// TIA Portal V17 export
// export: Created 2025-03-05T08:03:12.1647965Z, ExportSetting WithDefaults, DisplayName Totally Integrated Automation Portal, DisplayVersion V17 Update 8, DisplayName TIA Portal Openness, DisplayVersion V17 Update 8, DisplayName TIA Portal Version Control Interface, DisplayVersion V17, DisplayName SINAMICS Startdrive Advanced, DisplayVersion V17 SP2, DisplayName SINAMICS Startdrive G110M, G120, G120C, G120D, G120P, G115D, DisplayVersion V17 SP2, DisplayName SINAMICS Startdrive G130, G150, S120, S150, SINAMICS MV, S210, DisplayVersion V17 SP2, DisplayName STEP 7 Professional, DisplayVersion V17 Update 8, DisplayName SINUMERIK ONE STEP 7 Toolbox, DisplayVersion V17 Update 12, DisplayName SINUMERIK 840D sl STEP 7 Toolbox, DisplayVersion V17 Update 12, DisplayName STEP 7 Safety, DisplayVersion V17 Update 6, DisplayName WinCC Advanced, DisplayVersion V17 Update 8
FUNCTION "FC22100_HOPPER_SYSTEM_SENSORS" : Void   // FC22100, LAD
TITLE = FC22100 HOPPER SYSTEM SENSORS
{ S7_Optimized_Access := 'TRUE' }
VERSION : 0.1
// stored: AutoNumber false, IsIECCheckEnabled false, SetENOAutomatically false, UDAEnableTagReadback false
   VAR CONSTANT
      FC_NUMBER : UInt := 22100;
   END_VAR
   VAR_TEMP   // added for the SCL form of the ladder/FBD networks
      _w1 : Bool;
   END_VAR
BEGIN

REGION Network 1: /////_UNIT_01_SENSORS_/////
END_REGION

REGION Network 2: HOPPER 1 UNIT 01
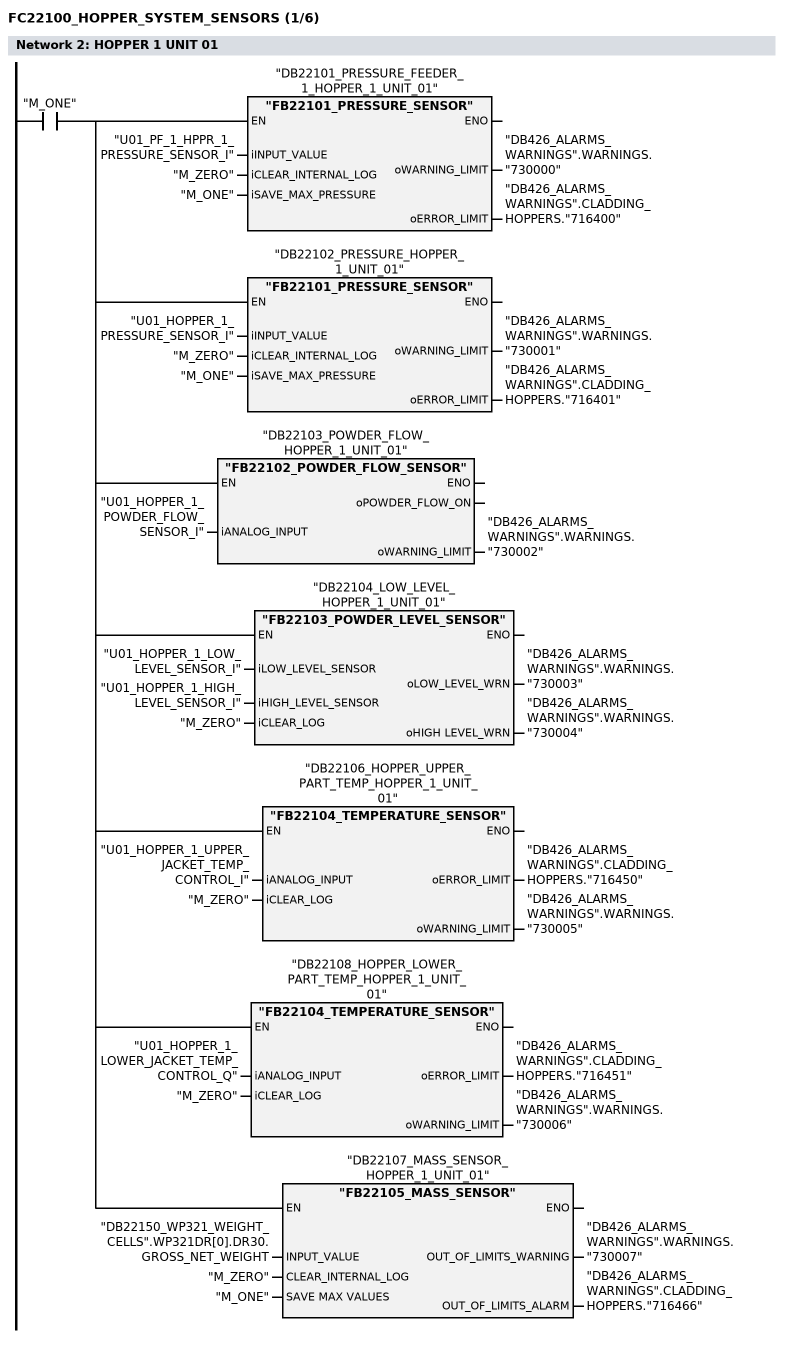
   RUNG wire#powerrail
      Contact( "M_ONE" )
      wire#w1
      "DB22101_PRESSURE_FEEDER_1_HOPPER_1_UNIT_01"(iINPUT_VALUE := "U01_PF_1_HPPR_1_PRESSURE_SENSOR_I", iCLEAR_INTERNAL_LOG := "M_ZERO", iSAVE_MAX_PRESSURE := "M_ONE", oWARNING_LIMIT => "DB426_ALARMS_WARNINGS".WARNINGS."730000", oERROR_LIMIT => "DB426_ALARMS_WARNINGS".CLADDING_HOPPERS."716400")
   END_RUNG
   RUNG wire#w1
      "DB22102_PRESSURE_HOPPER_1_UNIT_01"(iINPUT_VALUE := "U01_HOPPER_1_PRESSURE_SENSOR_I", iCLEAR_INTERNAL_LOG := "M_ZERO", iSAVE_MAX_PRESSURE := "M_ONE", oWARNING_LIMIT => "DB426_ALARMS_WARNINGS".WARNINGS."730001", oERROR_LIMIT => "DB426_ALARMS_WARNINGS".CLADDING_HOPPERS."716401")
   END_RUNG
   RUNG wire#w1
      "DB22103_POWDER_FLOW_HOPPER_1_UNIT_01"(iANALOG_INPUT := "U01_HOPPER_1_POWDER_FLOW_SENSOR_I", oPOWDER_FLOW_ON =>, oWARNING_LIMIT => "DB426_ALARMS_WARNINGS".WARNINGS."730002")
   END_RUNG
   RUNG wire#w1
      "DB22104_LOW_LEVEL_HOPPER_1_UNIT_01"(iLOW_LEVEL_SENSOR := "U01_HOPPER_1_LOW_LEVEL_SENSOR_I", iHIGH_LEVEL_SENSOR := "U01_HOPPER_1_HIGH_LEVEL_SENSOR_I", iCLEAR_LOG := "M_ZERO", oLOW_LEVEL_WRN => "DB426_ALARMS_WARNINGS".WARNINGS."730003", "oHIGH LEVEL_WRN" => "DB426_ALARMS_WARNINGS".WARNINGS."730004")
   END_RUNG
   RUNG wire#w1
      "DB22106_HOPPER_UPPER_PART_TEMP_HOPPER_1_UNIT_01"(iANALOG_INPUT := "U01_HOPPER_1_UPPER_JACKET_TEMP_CONTROL_I", iCLEAR_LOG := "M_ZERO", oERROR_LIMIT => "DB426_ALARMS_WARNINGS".CLADDING_HOPPERS."716450", oWARNING_LIMIT => "DB426_ALARMS_WARNINGS".WARNINGS."730005")
   END_RUNG
   RUNG wire#w1
      "DB22108_HOPPER_LOWER_PART_TEMP_HOPPER_1_UNIT_01"(iANALOG_INPUT := "U01_HOPPER_1_LOWER_JACKET_TEMP_CONTROL_Q", iCLEAR_LOG := "M_ZERO", oERROR_LIMIT => "DB426_ALARMS_WARNINGS".CLADDING_HOPPERS."716451", oWARNING_LIMIT => "DB426_ALARMS_WARNINGS".WARNINGS."730006")
   END_RUNG
   RUNG wire#w1
      "DB22107_MASS_SENSOR_HOPPER_1_UNIT_01"(INPUT_VALUE := "DB22150_WP321_WEIGHT_CELLS".WP321DR[0].DR30.GROSS_NET_WEIGHT, CLEAR_INTERNAL_LOG := "M_ZERO", "SAVE MAX VALUES" := "M_ONE", OUT_OF_LIMITS_WARNING => "DB426_ALARMS_WARNINGS".WARNINGS."730007", OUT_OF_LIMITS_ALARM => "DB426_ALARMS_WARNINGS".CLADDING_HOPPERS."716466")
   END_RUNG
   // the same network as SCL:
   #_w1 := "M_ONE";
   IF #_w1 THEN
       "DB22101_PRESSURE_FEEDER_1_HOPPER_1_UNIT_01"(iINPUT_VALUE := "U01_PF_1_HPPR_1_PRESSURE_SENSOR_I",   // "FB22101_PRESSURE_SENSOR"
                               iCLEAR_INTERNAL_LOG := "M_ZERO",
                               iSAVE_MAX_PRESSURE := "M_ONE",
                               oWARNING_LIMIT => "DB426_ALARMS_WARNINGS".WARNINGS."730000",
                               oERROR_LIMIT => "DB426_ALARMS_WARNINGS".CLADDING_HOPPERS."716400");
       "DB22102_PRESSURE_HOPPER_1_UNIT_01"(iINPUT_VALUE := "U01_HOPPER_1_PRESSURE_SENSOR_I",   // "FB22101_PRESSURE_SENSOR"
                               iCLEAR_INTERNAL_LOG := "M_ZERO",
                               iSAVE_MAX_PRESSURE := "M_ONE",
                               oWARNING_LIMIT => "DB426_ALARMS_WARNINGS".WARNINGS."730001",
                               oERROR_LIMIT => "DB426_ALARMS_WARNINGS".CLADDING_HOPPERS."716401");
       "DB22103_POWDER_FLOW_HOPPER_1_UNIT_01"(iANALOG_INPUT := "U01_HOPPER_1_POWDER_FLOW_SENSOR_I",   // "FB22102_POWDER_FLOW_SENSOR"
                               oWARNING_LIMIT => "DB426_ALARMS_WARNINGS".WARNINGS."730002");
       "DB22104_LOW_LEVEL_HOPPER_1_UNIT_01"(iLOW_LEVEL_SENSOR := "U01_HOPPER_1_LOW_LEVEL_SENSOR_I",   // "FB22103_POWDER_LEVEL_SENSOR"
                               iHIGH_LEVEL_SENSOR := "U01_HOPPER_1_HIGH_LEVEL_SENSOR_I",
                               iCLEAR_LOG := "M_ZERO",
                               oLOW_LEVEL_WRN => "DB426_ALARMS_WARNINGS".WARNINGS."730003",
                               "oHIGH LEVEL_WRN" => "DB426_ALARMS_WARNINGS".WARNINGS."730004");
       "DB22106_HOPPER_UPPER_PART_TEMP_HOPPER_1_UNIT_01"(iANALOG_INPUT := "U01_HOPPER_1_UPPER_JACKET_TEMP_CONTROL_I",   // "FB22104_TEMPERATURE_SENSOR"
                               iCLEAR_LOG := "M_ZERO",
                               oERROR_LIMIT => "DB426_ALARMS_WARNINGS".CLADDING_HOPPERS."716450",
                               oWARNING_LIMIT => "DB426_ALARMS_WARNINGS".WARNINGS."730005");
       "DB22108_HOPPER_LOWER_PART_TEMP_HOPPER_1_UNIT_01"(iANALOG_INPUT := "U01_HOPPER_1_LOWER_JACKET_TEMP_CONTROL_Q",   // "FB22104_TEMPERATURE_SENSOR"
                               iCLEAR_LOG := "M_ZERO",
                               oERROR_LIMIT => "DB426_ALARMS_WARNINGS".CLADDING_HOPPERS."716451",
                               oWARNING_LIMIT => "DB426_ALARMS_WARNINGS".WARNINGS."730006");
       "DB22107_MASS_SENSOR_HOPPER_1_UNIT_01"(INPUT_VALUE := "DB22150_WP321_WEIGHT_CELLS".WP321DR[0].DR30.GROSS_NET_WEIGHT,   // "FB22105_MASS_SENSOR"
                               CLEAR_INTERNAL_LOG := "M_ZERO",
                               "SAVE MAX VALUES" := "M_ONE",
                               OUT_OF_LIMITS_WARNING => "DB426_ALARMS_WARNINGS".WARNINGS."730007",
                               OUT_OF_LIMITS_ALARM => "DB426_ALARMS_WARNINGS".CLADDING_HOPPERS."716466");
   END_IF;
END_REGION

REGION Network 3: HOPPER 2 UNIT 01
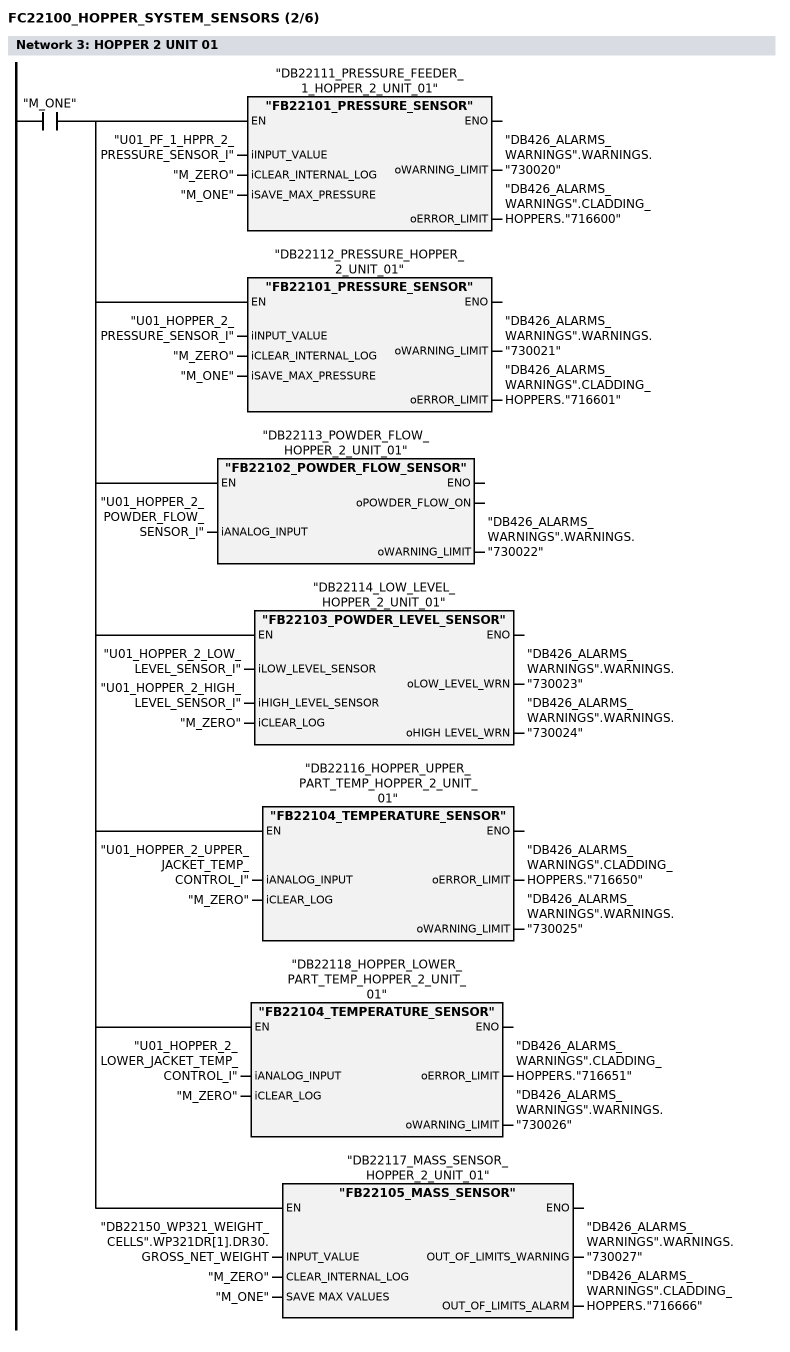
   RUNG wire#powerrail
      Contact( "M_ONE" )
      wire#w1
      "DB22111_PRESSURE_FEEDER_1_HOPPER_2_UNIT_01"(iINPUT_VALUE := "U01_PF_1_HPPR_2_PRESSURE_SENSOR_I", iCLEAR_INTERNAL_LOG := "M_ZERO", iSAVE_MAX_PRESSURE := "M_ONE", oWARNING_LIMIT => "DB426_ALARMS_WARNINGS".WARNINGS."730020", oERROR_LIMIT => "DB426_ALARMS_WARNINGS".CLADDING_HOPPERS."716600")
   END_RUNG
   RUNG wire#w1
      "DB22112_PRESSURE_HOPPER_2_UNIT_01"(iINPUT_VALUE := "U01_HOPPER_2_PRESSURE_SENSOR_I", iCLEAR_INTERNAL_LOG := "M_ZERO", iSAVE_MAX_PRESSURE := "M_ONE", oWARNING_LIMIT => "DB426_ALARMS_WARNINGS".WARNINGS."730021", oERROR_LIMIT => "DB426_ALARMS_WARNINGS".CLADDING_HOPPERS."716601")
   END_RUNG
   RUNG wire#w1
      "DB22113_POWDER_FLOW_HOPPER_2_UNIT_01"(iANALOG_INPUT := "U01_HOPPER_2_POWDER_FLOW_SENSOR_I", oPOWDER_FLOW_ON =>, oWARNING_LIMIT => "DB426_ALARMS_WARNINGS".WARNINGS."730022")
   END_RUNG
   RUNG wire#w1
      "DB22114_LOW_LEVEL_HOPPER_2_UNIT_01"(iLOW_LEVEL_SENSOR := "U01_HOPPER_2_LOW_LEVEL_SENSOR_I", iHIGH_LEVEL_SENSOR := "U01_HOPPER_2_HIGH_LEVEL_SENSOR_I", iCLEAR_LOG := "M_ZERO", oLOW_LEVEL_WRN => "DB426_ALARMS_WARNINGS".WARNINGS."730023", "oHIGH LEVEL_WRN" => "DB426_ALARMS_WARNINGS".WARNINGS."730024")
   END_RUNG
   RUNG wire#w1
      "DB22116_HOPPER_UPPER_PART_TEMP_HOPPER_2_UNIT_01"(iANALOG_INPUT := "U01_HOPPER_2_UPPER_JACKET_TEMP_CONTROL_I", iCLEAR_LOG := "M_ZERO", oERROR_LIMIT => "DB426_ALARMS_WARNINGS".CLADDING_HOPPERS."716650", oWARNING_LIMIT => "DB426_ALARMS_WARNINGS".WARNINGS."730025")
   END_RUNG
   RUNG wire#w1
      "DB22118_HOPPER_LOWER_PART_TEMP_HOPPER_2_UNIT_01"(iANALOG_INPUT := "U01_HOPPER_2_LOWER_JACKET_TEMP_CONTROL_I", iCLEAR_LOG := "M_ZERO", oERROR_LIMIT => "DB426_ALARMS_WARNINGS".CLADDING_HOPPERS."716651", oWARNING_LIMIT => "DB426_ALARMS_WARNINGS".WARNINGS."730026")
   END_RUNG
   RUNG wire#w1
      "DB22117_MASS_SENSOR_HOPPER_2_UNIT_01"(INPUT_VALUE := "DB22150_WP321_WEIGHT_CELLS".WP321DR[1].DR30.GROSS_NET_WEIGHT, CLEAR_INTERNAL_LOG := "M_ZERO", "SAVE MAX VALUES" := "M_ONE", OUT_OF_LIMITS_WARNING => "DB426_ALARMS_WARNINGS".WARNINGS."730027", OUT_OF_LIMITS_ALARM => "DB426_ALARMS_WARNINGS".CLADDING_HOPPERS."716666")
   END_RUNG
   // the same network as SCL:
   #_w1 := "M_ONE";
   IF #_w1 THEN
       "DB22111_PRESSURE_FEEDER_1_HOPPER_2_UNIT_01"(iINPUT_VALUE := "U01_PF_1_HPPR_2_PRESSURE_SENSOR_I",   // "FB22101_PRESSURE_SENSOR"
                               iCLEAR_INTERNAL_LOG := "M_ZERO",
                               iSAVE_MAX_PRESSURE := "M_ONE",
                               oWARNING_LIMIT => "DB426_ALARMS_WARNINGS".WARNINGS."730020",
                               oERROR_LIMIT => "DB426_ALARMS_WARNINGS".CLADDING_HOPPERS."716600");
       "DB22112_PRESSURE_HOPPER_2_UNIT_01"(iINPUT_VALUE := "U01_HOPPER_2_PRESSURE_SENSOR_I",   // "FB22101_PRESSURE_SENSOR"
                               iCLEAR_INTERNAL_LOG := "M_ZERO",
                               iSAVE_MAX_PRESSURE := "M_ONE",
                               oWARNING_LIMIT => "DB426_ALARMS_WARNINGS".WARNINGS."730021",
                               oERROR_LIMIT => "DB426_ALARMS_WARNINGS".CLADDING_HOPPERS."716601");
       "DB22113_POWDER_FLOW_HOPPER_2_UNIT_01"(iANALOG_INPUT := "U01_HOPPER_2_POWDER_FLOW_SENSOR_I",   // "FB22102_POWDER_FLOW_SENSOR"
                               oWARNING_LIMIT => "DB426_ALARMS_WARNINGS".WARNINGS."730022");
       "DB22114_LOW_LEVEL_HOPPER_2_UNIT_01"(iLOW_LEVEL_SENSOR := "U01_HOPPER_2_LOW_LEVEL_SENSOR_I",   // "FB22103_POWDER_LEVEL_SENSOR"
                               iHIGH_LEVEL_SENSOR := "U01_HOPPER_2_HIGH_LEVEL_SENSOR_I",
                               iCLEAR_LOG := "M_ZERO",
                               oLOW_LEVEL_WRN => "DB426_ALARMS_WARNINGS".WARNINGS."730023",
                               "oHIGH LEVEL_WRN" => "DB426_ALARMS_WARNINGS".WARNINGS."730024");
       "DB22116_HOPPER_UPPER_PART_TEMP_HOPPER_2_UNIT_01"(iANALOG_INPUT := "U01_HOPPER_2_UPPER_JACKET_TEMP_CONTROL_I",   // "FB22104_TEMPERATURE_SENSOR"
                               iCLEAR_LOG := "M_ZERO",
                               oERROR_LIMIT => "DB426_ALARMS_WARNINGS".CLADDING_HOPPERS."716650",
                               oWARNING_LIMIT => "DB426_ALARMS_WARNINGS".WARNINGS."730025");
       "DB22118_HOPPER_LOWER_PART_TEMP_HOPPER_2_UNIT_01"(iANALOG_INPUT := "U01_HOPPER_2_LOWER_JACKET_TEMP_CONTROL_I",   // "FB22104_TEMPERATURE_SENSOR"
                               iCLEAR_LOG := "M_ZERO",
                               oERROR_LIMIT => "DB426_ALARMS_WARNINGS".CLADDING_HOPPERS."716651",
                               oWARNING_LIMIT => "DB426_ALARMS_WARNINGS".WARNINGS."730026");
       "DB22117_MASS_SENSOR_HOPPER_2_UNIT_01"(INPUT_VALUE := "DB22150_WP321_WEIGHT_CELLS".WP321DR[1].DR30.GROSS_NET_WEIGHT,   // "FB22105_MASS_SENSOR"
                               CLEAR_INTERNAL_LOG := "M_ZERO",
                               "SAVE MAX VALUES" := "M_ONE",
                               OUT_OF_LIMITS_WARNING => "DB426_ALARMS_WARNINGS".WARNINGS."730027",
                               OUT_OF_LIMITS_ALARM => "DB426_ALARMS_WARNINGS".CLADDING_HOPPERS."716666");
   END_IF;
END_REGION

REGION Network 4: /////_UNIT_02_SENSORS_/////
END_REGION

REGION Network 5: HOPPER 1 UNIT 02
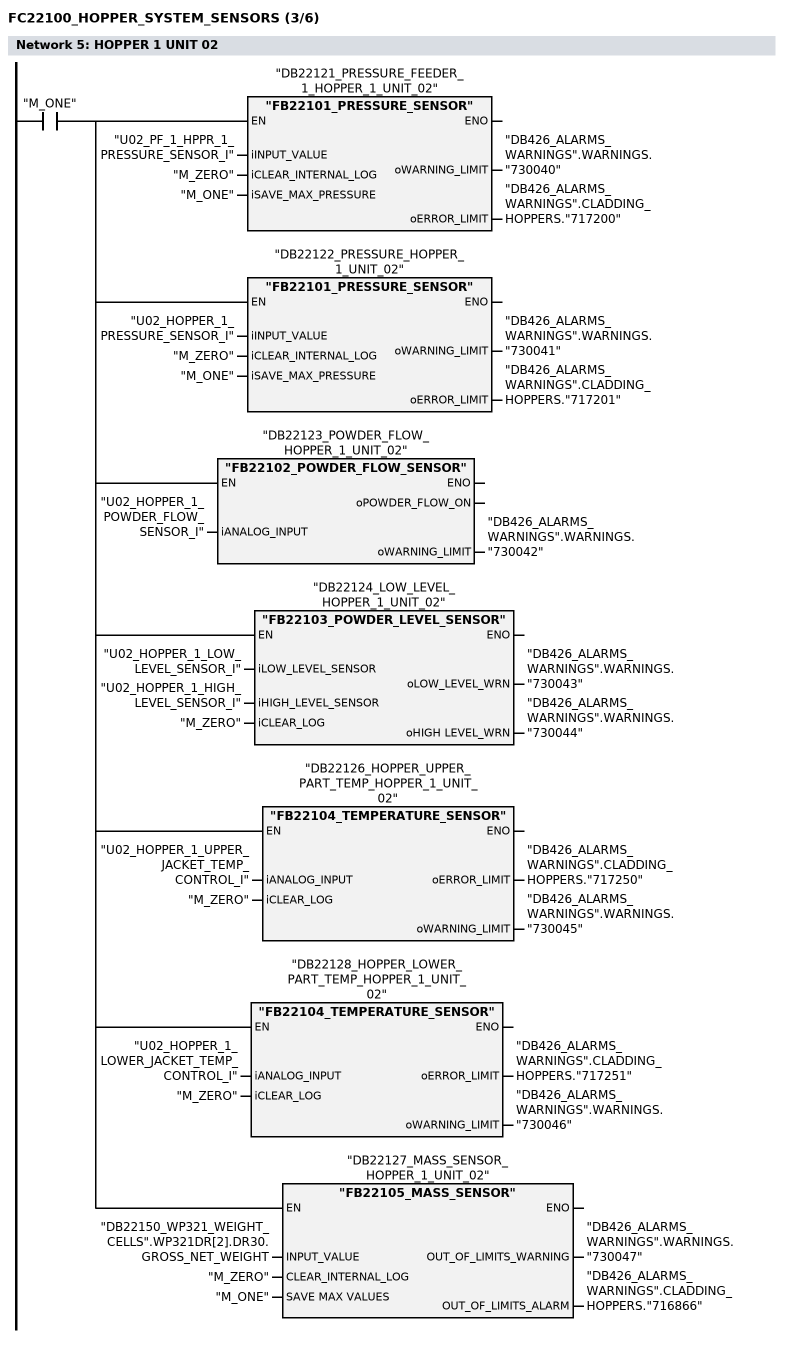
   RUNG wire#powerrail
      Contact( "M_ONE" )
      wire#w1
      "DB22121_PRESSURE_FEEDER_1_HOPPER_1_UNIT_02"(iINPUT_VALUE := "U02_PF_1_HPPR_1_PRESSURE_SENSOR_I", iCLEAR_INTERNAL_LOG := "M_ZERO", iSAVE_MAX_PRESSURE := "M_ONE", oWARNING_LIMIT => "DB426_ALARMS_WARNINGS".WARNINGS."730040", oERROR_LIMIT => "DB426_ALARMS_WARNINGS".CLADDING_HOPPERS."717200")
   END_RUNG
   RUNG wire#w1
      "DB22122_PRESSURE_HOPPER_1_UNIT_02"(iINPUT_VALUE := "U02_HOPPER_1_PRESSURE_SENSOR_I", iCLEAR_INTERNAL_LOG := "M_ZERO", iSAVE_MAX_PRESSURE := "M_ONE", oWARNING_LIMIT => "DB426_ALARMS_WARNINGS".WARNINGS."730041", oERROR_LIMIT => "DB426_ALARMS_WARNINGS".CLADDING_HOPPERS."717201")
   END_RUNG
   RUNG wire#w1
      "DB22123_POWDER_FLOW_HOPPER_1_UNIT_02"(iANALOG_INPUT := "U02_HOPPER_1_POWDER_FLOW_SENSOR_I", oPOWDER_FLOW_ON =>, oWARNING_LIMIT => "DB426_ALARMS_WARNINGS".WARNINGS."730042")
   END_RUNG
   RUNG wire#w1
      "DB22124_LOW_LEVEL_HOPPER_1_UNIT_02"(iLOW_LEVEL_SENSOR := "U02_HOPPER_1_LOW_LEVEL_SENSOR_I", iHIGH_LEVEL_SENSOR := "U02_HOPPER_1_HIGH_LEVEL_SENSOR_I", iCLEAR_LOG := "M_ZERO", oLOW_LEVEL_WRN => "DB426_ALARMS_WARNINGS".WARNINGS."730043", "oHIGH LEVEL_WRN" => "DB426_ALARMS_WARNINGS".WARNINGS."730044")
   END_RUNG
   RUNG wire#w1
      "DB22126_HOPPER_UPPER_PART_TEMP_HOPPER_1_UNIT_02"(iANALOG_INPUT := "U02_HOPPER_1_UPPER_JACKET_TEMP_CONTROL_I", iCLEAR_LOG := "M_ZERO", oERROR_LIMIT => "DB426_ALARMS_WARNINGS".CLADDING_HOPPERS."717250", oWARNING_LIMIT => "DB426_ALARMS_WARNINGS".WARNINGS."730045")
   END_RUNG
   RUNG wire#w1
      "DB22128_HOPPER_LOWER_PART_TEMP_HOPPER_1_UNIT_02"(iANALOG_INPUT := "U02_HOPPER_1_LOWER_JACKET_TEMP_CONTROL_I", iCLEAR_LOG := "M_ZERO", oERROR_LIMIT => "DB426_ALARMS_WARNINGS".CLADDING_HOPPERS."717251", oWARNING_LIMIT => "DB426_ALARMS_WARNINGS".WARNINGS."730046")
   END_RUNG
   RUNG wire#w1
      "DB22127_MASS_SENSOR_HOPPER_1_UNIT_02"(INPUT_VALUE := "DB22150_WP321_WEIGHT_CELLS".WP321DR[2].DR30.GROSS_NET_WEIGHT, CLEAR_INTERNAL_LOG := "M_ZERO", "SAVE MAX VALUES" := "M_ONE", OUT_OF_LIMITS_WARNING => "DB426_ALARMS_WARNINGS".WARNINGS."730047", OUT_OF_LIMITS_ALARM => "DB426_ALARMS_WARNINGS".CLADDING_HOPPERS."716866")
   END_RUNG
   // the same network as SCL:
   #_w1 := "M_ONE";
   IF #_w1 THEN
       "DB22121_PRESSURE_FEEDER_1_HOPPER_1_UNIT_02"(iINPUT_VALUE := "U02_PF_1_HPPR_1_PRESSURE_SENSOR_I",   // "FB22101_PRESSURE_SENSOR"
                               iCLEAR_INTERNAL_LOG := "M_ZERO",
                               iSAVE_MAX_PRESSURE := "M_ONE",
                               oWARNING_LIMIT => "DB426_ALARMS_WARNINGS".WARNINGS."730040",
                               oERROR_LIMIT => "DB426_ALARMS_WARNINGS".CLADDING_HOPPERS."717200");
       "DB22122_PRESSURE_HOPPER_1_UNIT_02"(iINPUT_VALUE := "U02_HOPPER_1_PRESSURE_SENSOR_I",   // "FB22101_PRESSURE_SENSOR"
                               iCLEAR_INTERNAL_LOG := "M_ZERO",
                               iSAVE_MAX_PRESSURE := "M_ONE",
                               oWARNING_LIMIT => "DB426_ALARMS_WARNINGS".WARNINGS."730041",
                               oERROR_LIMIT => "DB426_ALARMS_WARNINGS".CLADDING_HOPPERS."717201");
       "DB22123_POWDER_FLOW_HOPPER_1_UNIT_02"(iANALOG_INPUT := "U02_HOPPER_1_POWDER_FLOW_SENSOR_I",   // "FB22102_POWDER_FLOW_SENSOR"
                               oWARNING_LIMIT => "DB426_ALARMS_WARNINGS".WARNINGS."730042");
       "DB22124_LOW_LEVEL_HOPPER_1_UNIT_02"(iLOW_LEVEL_SENSOR := "U02_HOPPER_1_LOW_LEVEL_SENSOR_I",   // "FB22103_POWDER_LEVEL_SENSOR"
                               iHIGH_LEVEL_SENSOR := "U02_HOPPER_1_HIGH_LEVEL_SENSOR_I",
                               iCLEAR_LOG := "M_ZERO",
                               oLOW_LEVEL_WRN => "DB426_ALARMS_WARNINGS".WARNINGS."730043",
                               "oHIGH LEVEL_WRN" => "DB426_ALARMS_WARNINGS".WARNINGS."730044");
       "DB22126_HOPPER_UPPER_PART_TEMP_HOPPER_1_UNIT_02"(iANALOG_INPUT := "U02_HOPPER_1_UPPER_JACKET_TEMP_CONTROL_I",   // "FB22104_TEMPERATURE_SENSOR"
                               iCLEAR_LOG := "M_ZERO",
                               oERROR_LIMIT => "DB426_ALARMS_WARNINGS".CLADDING_HOPPERS."717250",
                               oWARNING_LIMIT => "DB426_ALARMS_WARNINGS".WARNINGS."730045");
       "DB22128_HOPPER_LOWER_PART_TEMP_HOPPER_1_UNIT_02"(iANALOG_INPUT := "U02_HOPPER_1_LOWER_JACKET_TEMP_CONTROL_I",   // "FB22104_TEMPERATURE_SENSOR"
                               iCLEAR_LOG := "M_ZERO",
                               oERROR_LIMIT => "DB426_ALARMS_WARNINGS".CLADDING_HOPPERS."717251",
                               oWARNING_LIMIT => "DB426_ALARMS_WARNINGS".WARNINGS."730046");
       "DB22127_MASS_SENSOR_HOPPER_1_UNIT_02"(INPUT_VALUE := "DB22150_WP321_WEIGHT_CELLS".WP321DR[2].DR30.GROSS_NET_WEIGHT,   // "FB22105_MASS_SENSOR"
                               CLEAR_INTERNAL_LOG := "M_ZERO",
                               "SAVE MAX VALUES" := "M_ONE",
                               OUT_OF_LIMITS_WARNING => "DB426_ALARMS_WARNINGS".WARNINGS."730047",
                               OUT_OF_LIMITS_ALARM => "DB426_ALARMS_WARNINGS".CLADDING_HOPPERS."716866");
   END_IF;
END_REGION

REGION Network 6: HOPPER 2 UNIT 02
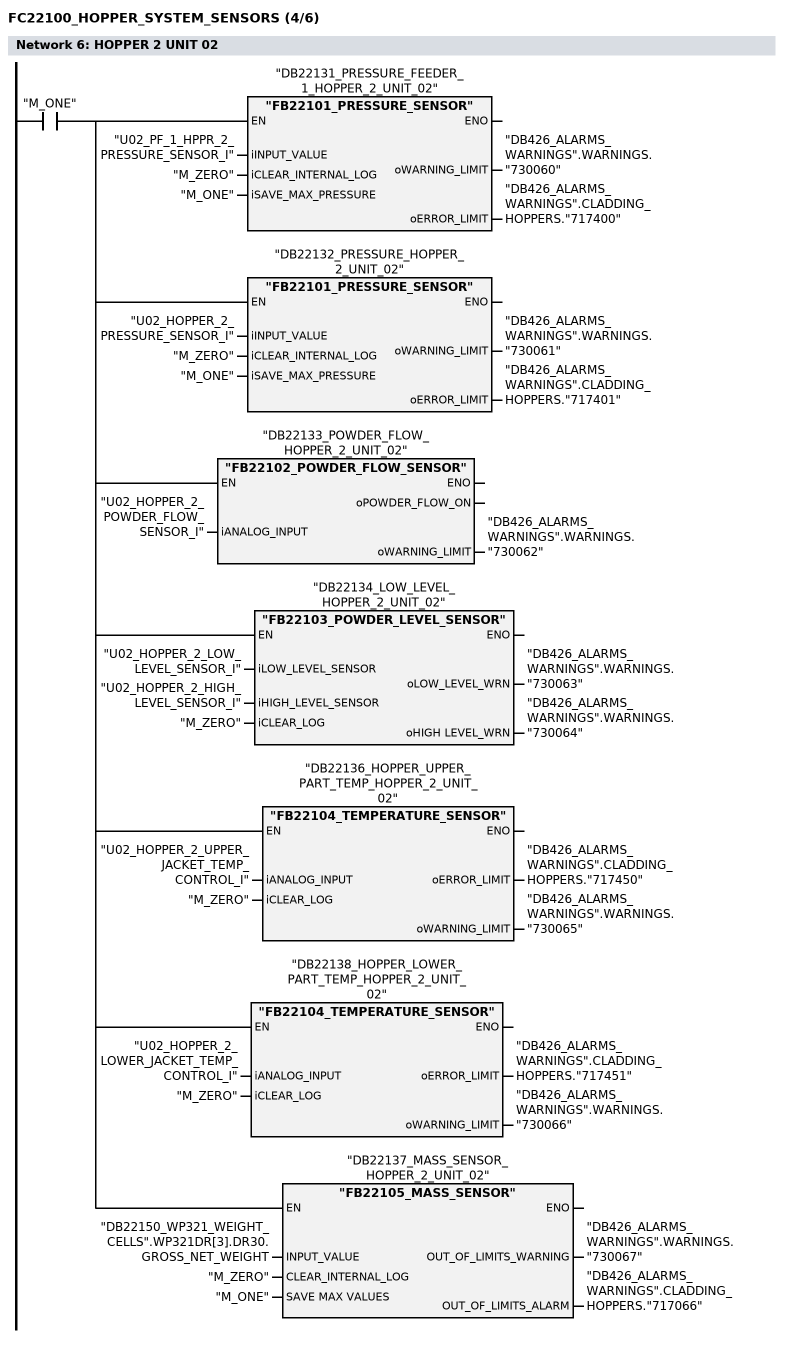
   RUNG wire#powerrail
      Contact( "M_ONE" )
      wire#w1
      "DB22131_PRESSURE_FEEDER_1_HOPPER_2_UNIT_02"(iINPUT_VALUE := "U02_PF_1_HPPR_2_PRESSURE_SENSOR_I", iCLEAR_INTERNAL_LOG := "M_ZERO", iSAVE_MAX_PRESSURE := "M_ONE", oWARNING_LIMIT => "DB426_ALARMS_WARNINGS".WARNINGS."730060", oERROR_LIMIT => "DB426_ALARMS_WARNINGS".CLADDING_HOPPERS."717400")
   END_RUNG
   RUNG wire#w1
      "DB22132_PRESSURE_HOPPER_2_UNIT_02"(iINPUT_VALUE := "U02_HOPPER_2_PRESSURE_SENSOR_I", iCLEAR_INTERNAL_LOG := "M_ZERO", iSAVE_MAX_PRESSURE := "M_ONE", oWARNING_LIMIT => "DB426_ALARMS_WARNINGS".WARNINGS."730061", oERROR_LIMIT => "DB426_ALARMS_WARNINGS".CLADDING_HOPPERS."717401")
   END_RUNG
   RUNG wire#w1
      "DB22133_POWDER_FLOW_HOPPER_2_UNIT_02"(iANALOG_INPUT := "U02_HOPPER_2_POWDER_FLOW_SENSOR_I", oPOWDER_FLOW_ON =>, oWARNING_LIMIT => "DB426_ALARMS_WARNINGS".WARNINGS."730062")
   END_RUNG
   RUNG wire#w1
      "DB22134_LOW_LEVEL_HOPPER_2_UNIT_02"(iLOW_LEVEL_SENSOR := "U02_HOPPER_2_LOW_LEVEL_SENSOR_I", iHIGH_LEVEL_SENSOR := "U02_HOPPER_2_HIGH_LEVEL_SENSOR_I", iCLEAR_LOG := "M_ZERO", oLOW_LEVEL_WRN => "DB426_ALARMS_WARNINGS".WARNINGS."730063", "oHIGH LEVEL_WRN" => "DB426_ALARMS_WARNINGS".WARNINGS."730064")
   END_RUNG
   RUNG wire#w1
      "DB22136_HOPPER_UPPER_PART_TEMP_HOPPER_2_UNIT_02"(iANALOG_INPUT := "U02_HOPPER_2_UPPER_JACKET_TEMP_CONTROL_I", iCLEAR_LOG := "M_ZERO", oERROR_LIMIT => "DB426_ALARMS_WARNINGS".CLADDING_HOPPERS."717450", oWARNING_LIMIT => "DB426_ALARMS_WARNINGS".WARNINGS."730065")
   END_RUNG
   RUNG wire#w1
      "DB22138_HOPPER_LOWER_PART_TEMP_HOPPER_2_UNIT_02"(iANALOG_INPUT := "U02_HOPPER_2_LOWER_JACKET_TEMP_CONTROL_I", iCLEAR_LOG := "M_ZERO", oERROR_LIMIT => "DB426_ALARMS_WARNINGS".CLADDING_HOPPERS."717451", oWARNING_LIMIT => "DB426_ALARMS_WARNINGS".WARNINGS."730066")
   END_RUNG
   RUNG wire#w1
      "DB22137_MASS_SENSOR_HOPPER_2_UNIT_02"(INPUT_VALUE := "DB22150_WP321_WEIGHT_CELLS".WP321DR[3].DR30.GROSS_NET_WEIGHT, CLEAR_INTERNAL_LOG := "M_ZERO", "SAVE MAX VALUES" := "M_ONE", OUT_OF_LIMITS_WARNING => "DB426_ALARMS_WARNINGS".WARNINGS."730067", OUT_OF_LIMITS_ALARM => "DB426_ALARMS_WARNINGS".CLADDING_HOPPERS."717066")
   END_RUNG
   // the same network as SCL:
   #_w1 := "M_ONE";
   IF #_w1 THEN
       "DB22131_PRESSURE_FEEDER_1_HOPPER_2_UNIT_02"(iINPUT_VALUE := "U02_PF_1_HPPR_2_PRESSURE_SENSOR_I",   // "FB22101_PRESSURE_SENSOR"
                               iCLEAR_INTERNAL_LOG := "M_ZERO",
                               iSAVE_MAX_PRESSURE := "M_ONE",
                               oWARNING_LIMIT => "DB426_ALARMS_WARNINGS".WARNINGS."730060",
                               oERROR_LIMIT => "DB426_ALARMS_WARNINGS".CLADDING_HOPPERS."717400");
       "DB22132_PRESSURE_HOPPER_2_UNIT_02"(iINPUT_VALUE := "U02_HOPPER_2_PRESSURE_SENSOR_I",   // "FB22101_PRESSURE_SENSOR"
                               iCLEAR_INTERNAL_LOG := "M_ZERO",
                               iSAVE_MAX_PRESSURE := "M_ONE",
                               oWARNING_LIMIT => "DB426_ALARMS_WARNINGS".WARNINGS."730061",
                               oERROR_LIMIT => "DB426_ALARMS_WARNINGS".CLADDING_HOPPERS."717401");
       "DB22133_POWDER_FLOW_HOPPER_2_UNIT_02"(iANALOG_INPUT := "U02_HOPPER_2_POWDER_FLOW_SENSOR_I",   // "FB22102_POWDER_FLOW_SENSOR"
                               oWARNING_LIMIT => "DB426_ALARMS_WARNINGS".WARNINGS."730062");
       "DB22134_LOW_LEVEL_HOPPER_2_UNIT_02"(iLOW_LEVEL_SENSOR := "U02_HOPPER_2_LOW_LEVEL_SENSOR_I",   // "FB22103_POWDER_LEVEL_SENSOR"
                               iHIGH_LEVEL_SENSOR := "U02_HOPPER_2_HIGH_LEVEL_SENSOR_I",
                               iCLEAR_LOG := "M_ZERO",
                               oLOW_LEVEL_WRN => "DB426_ALARMS_WARNINGS".WARNINGS."730063",
                               "oHIGH LEVEL_WRN" => "DB426_ALARMS_WARNINGS".WARNINGS."730064");
       "DB22136_HOPPER_UPPER_PART_TEMP_HOPPER_2_UNIT_02"(iANALOG_INPUT := "U02_HOPPER_2_UPPER_JACKET_TEMP_CONTROL_I",   // "FB22104_TEMPERATURE_SENSOR"
                               iCLEAR_LOG := "M_ZERO",
                               oERROR_LIMIT => "DB426_ALARMS_WARNINGS".CLADDING_HOPPERS."717450",
                               oWARNING_LIMIT => "DB426_ALARMS_WARNINGS".WARNINGS."730065");
       "DB22138_HOPPER_LOWER_PART_TEMP_HOPPER_2_UNIT_02"(iANALOG_INPUT := "U02_HOPPER_2_LOWER_JACKET_TEMP_CONTROL_I",   // "FB22104_TEMPERATURE_SENSOR"
                               iCLEAR_LOG := "M_ZERO",
                               oERROR_LIMIT => "DB426_ALARMS_WARNINGS".CLADDING_HOPPERS."717451",
                               oWARNING_LIMIT => "DB426_ALARMS_WARNINGS".WARNINGS."730066");
       "DB22137_MASS_SENSOR_HOPPER_2_UNIT_02"(INPUT_VALUE := "DB22150_WP321_WEIGHT_CELLS".WP321DR[3].DR30.GROSS_NET_WEIGHT,   // "FB22105_MASS_SENSOR"
                               CLEAR_INTERNAL_LOG := "M_ZERO",
                               "SAVE MAX VALUES" := "M_ONE",
                               OUT_OF_LIMITS_WARNING => "DB426_ALARMS_WARNINGS".WARNINGS."730067",
                               OUT_OF_LIMITS_ALARM => "DB426_ALARMS_WARNINGS".CLADDING_HOPPERS."717066");
   END_IF;
END_REGION

REGION Network 7: HOPPER 3 UNIT 02
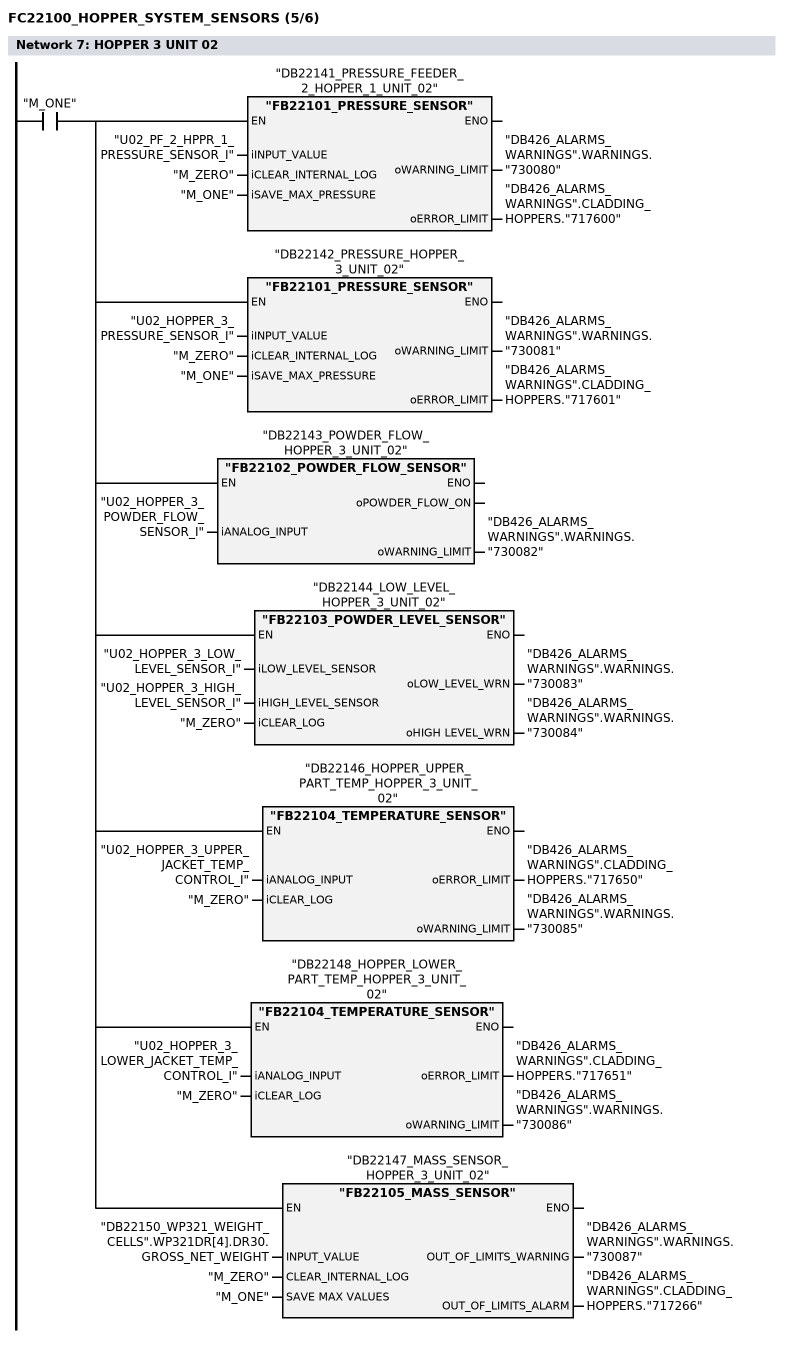
   RUNG wire#powerrail
      Contact( "M_ONE" )
      wire#w1
      "DB22141_PRESSURE_FEEDER_2_HOPPER_1_UNIT_02"(iINPUT_VALUE := "U02_PF_2_HPPR_1_PRESSURE_SENSOR_I", iCLEAR_INTERNAL_LOG := "M_ZERO", iSAVE_MAX_PRESSURE := "M_ONE", oWARNING_LIMIT => "DB426_ALARMS_WARNINGS".WARNINGS."730080", oERROR_LIMIT => "DB426_ALARMS_WARNINGS".CLADDING_HOPPERS."717600")
   END_RUNG
   RUNG wire#w1
      "DB22142_PRESSURE_HOPPER_3_UNIT_02"(iINPUT_VALUE := "U02_HOPPER_3_PRESSURE_SENSOR_I", iCLEAR_INTERNAL_LOG := "M_ZERO", iSAVE_MAX_PRESSURE := "M_ONE", oWARNING_LIMIT => "DB426_ALARMS_WARNINGS".WARNINGS."730081", oERROR_LIMIT => "DB426_ALARMS_WARNINGS".CLADDING_HOPPERS."717601")
   END_RUNG
   RUNG wire#w1
      "DB22143_POWDER_FLOW_HOPPER_3_UNIT_02"(iANALOG_INPUT := "U02_HOPPER_3_POWDER_FLOW_SENSOR_I", oPOWDER_FLOW_ON =>, oWARNING_LIMIT => "DB426_ALARMS_WARNINGS".WARNINGS."730082")
   END_RUNG
   RUNG wire#w1
      "DB22144_LOW_LEVEL_HOPPER_3_UNIT_02"(iLOW_LEVEL_SENSOR := "U02_HOPPER_3_LOW_LEVEL_SENSOR_I", iHIGH_LEVEL_SENSOR := "U02_HOPPER_3_HIGH_LEVEL_SENSOR_I", iCLEAR_LOG := "M_ZERO", oLOW_LEVEL_WRN => "DB426_ALARMS_WARNINGS".WARNINGS."730083", "oHIGH LEVEL_WRN" => "DB426_ALARMS_WARNINGS".WARNINGS."730084")
   END_RUNG
   RUNG wire#w1
      "DB22146_HOPPER_UPPER_PART_TEMP_HOPPER_3_UNIT_02"(iANALOG_INPUT := "U02_HOPPER_3_UPPER_JACKET_TEMP_CONTROL_I", iCLEAR_LOG := "M_ZERO", oERROR_LIMIT => "DB426_ALARMS_WARNINGS".CLADDING_HOPPERS."717650", oWARNING_LIMIT => "DB426_ALARMS_WARNINGS".WARNINGS."730085")
   END_RUNG
   RUNG wire#w1
      "DB22148_HOPPER_LOWER_PART_TEMP_HOPPER_3_UNIT_02"(iANALOG_INPUT := "U02_HOPPER_3_LOWER_JACKET_TEMP_CONTROL_I", iCLEAR_LOG := "M_ZERO", oERROR_LIMIT => "DB426_ALARMS_WARNINGS".CLADDING_HOPPERS."717651", oWARNING_LIMIT => "DB426_ALARMS_WARNINGS".WARNINGS."730086")
   END_RUNG
   RUNG wire#w1
      "DB22147_MASS_SENSOR_HOPPER_3_UNIT_02"(INPUT_VALUE := "DB22150_WP321_WEIGHT_CELLS".WP321DR[4].DR30.GROSS_NET_WEIGHT, CLEAR_INTERNAL_LOG := "M_ZERO", "SAVE MAX VALUES" := "M_ONE", OUT_OF_LIMITS_WARNING => "DB426_ALARMS_WARNINGS".WARNINGS."730087", OUT_OF_LIMITS_ALARM => "DB426_ALARMS_WARNINGS".CLADDING_HOPPERS."717266")
   END_RUNG
   // the same network as SCL:
   #_w1 := "M_ONE";
   IF #_w1 THEN
       "DB22141_PRESSURE_FEEDER_2_HOPPER_1_UNIT_02"(iINPUT_VALUE := "U02_PF_2_HPPR_1_PRESSURE_SENSOR_I",   // "FB22101_PRESSURE_SENSOR"
                               iCLEAR_INTERNAL_LOG := "M_ZERO",
                               iSAVE_MAX_PRESSURE := "M_ONE",
                               oWARNING_LIMIT => "DB426_ALARMS_WARNINGS".WARNINGS."730080",
                               oERROR_LIMIT => "DB426_ALARMS_WARNINGS".CLADDING_HOPPERS."717600");
       "DB22142_PRESSURE_HOPPER_3_UNIT_02"(iINPUT_VALUE := "U02_HOPPER_3_PRESSURE_SENSOR_I",   // "FB22101_PRESSURE_SENSOR"
                               iCLEAR_INTERNAL_LOG := "M_ZERO",
                               iSAVE_MAX_PRESSURE := "M_ONE",
                               oWARNING_LIMIT => "DB426_ALARMS_WARNINGS".WARNINGS."730081",
                               oERROR_LIMIT => "DB426_ALARMS_WARNINGS".CLADDING_HOPPERS."717601");
       "DB22143_POWDER_FLOW_HOPPER_3_UNIT_02"(iANALOG_INPUT := "U02_HOPPER_3_POWDER_FLOW_SENSOR_I",   // "FB22102_POWDER_FLOW_SENSOR"
                               oWARNING_LIMIT => "DB426_ALARMS_WARNINGS".WARNINGS."730082");
       "DB22144_LOW_LEVEL_HOPPER_3_UNIT_02"(iLOW_LEVEL_SENSOR := "U02_HOPPER_3_LOW_LEVEL_SENSOR_I",   // "FB22103_POWDER_LEVEL_SENSOR"
                               iHIGH_LEVEL_SENSOR := "U02_HOPPER_3_HIGH_LEVEL_SENSOR_I",
                               iCLEAR_LOG := "M_ZERO",
                               oLOW_LEVEL_WRN => "DB426_ALARMS_WARNINGS".WARNINGS."730083",
                               "oHIGH LEVEL_WRN" => "DB426_ALARMS_WARNINGS".WARNINGS."730084");
       "DB22146_HOPPER_UPPER_PART_TEMP_HOPPER_3_UNIT_02"(iANALOG_INPUT := "U02_HOPPER_3_UPPER_JACKET_TEMP_CONTROL_I",   // "FB22104_TEMPERATURE_SENSOR"
                               iCLEAR_LOG := "M_ZERO",
                               oERROR_LIMIT => "DB426_ALARMS_WARNINGS".CLADDING_HOPPERS."717650",
                               oWARNING_LIMIT => "DB426_ALARMS_WARNINGS".WARNINGS."730085");
       "DB22148_HOPPER_LOWER_PART_TEMP_HOPPER_3_UNIT_02"(iANALOG_INPUT := "U02_HOPPER_3_LOWER_JACKET_TEMP_CONTROL_I",   // "FB22104_TEMPERATURE_SENSOR"
                               iCLEAR_LOG := "M_ZERO",
                               oERROR_LIMIT => "DB426_ALARMS_WARNINGS".CLADDING_HOPPERS."717651",
                               oWARNING_LIMIT => "DB426_ALARMS_WARNINGS".WARNINGS."730086");
       "DB22147_MASS_SENSOR_HOPPER_3_UNIT_02"(INPUT_VALUE := "DB22150_WP321_WEIGHT_CELLS".WP321DR[4].DR30.GROSS_NET_WEIGHT,   // "FB22105_MASS_SENSOR"
                               CLEAR_INTERNAL_LOG := "M_ZERO",
                               "SAVE MAX VALUES" := "M_ONE",
                               OUT_OF_LIMITS_WARNING => "DB426_ALARMS_WARNINGS".WARNINGS."730087",
                               OUT_OF_LIMITS_ALARM => "DB426_ALARMS_WARNINGS".CLADDING_HOPPERS."717266");
   END_IF;
END_REGION

REGION Network 8: CALL FB22108 WP321_MUL_CALL
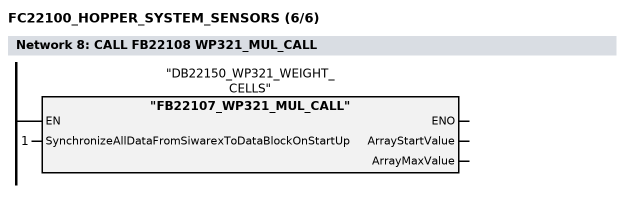
   RUNG wire#powerrail
      "DB22150_WP321_WEIGHT_CELLS"(SynchronizeAllDataFromSiwarexToDataBlockOnStartUp := 1, ArrayStartValue =>, ArrayMaxValue =>)
   END_RUNG
   // the same network as SCL:
   "DB22150_WP321_WEIGHT_CELLS"(SynchronizeAllDataFromSiwarexToDataBlockOnStartUp := 1);   // "FB22107_WP321_MUL_CALL"
END_REGION
END_FUNCTION
